PROGRAM MAIN
VAR
	tst_out : BYTE;
END_VAR


GVL_TEST.TST_OUT := tst_out;

END_PROGRAM

(* stored: Version 1.1.0.1, ProductVersion 3.1.4024.12
   POU MAIN: Id {371f4e99-333a-4563-9f26-aefdbf01b04d}, SpecialFunc None *)
